// TIA Portal V20 export
DATA_BLOCK "Config"   // DB102
// stored: Access Published, MemoryReserve 100, Namespace Unit1.Em5
   VAR
      em : "LAF_typeEmConfiguration";   // Configuration of EM Parameters
      axis : Array[1.._.U1EM5_NO_OF_AXES] of DB_ANY;
      moduleAccessPoint : Array[1.._.U1EM5_NO_OF_AXES] of HW_SUBMODULE;
   END_VAR
   VAR RETAIN
      cmNgAndManualInputAxisY : "LBC_typeAxis64PosConfiguration";
      cmMagazineAxisZ : "LBC_typeAxis64PosConfiguration";
      cmNgAndManualInputCylinderUpDown : "LBC_typeTwoWayActuatorConfiguration";
      cmNgAndManualInputVacuum1OnOff : "LBC_typeTwoWayActuatorConfiguration";
      cmNgAndManualInputVacuum2OnOff : "LBC_typeTwoWayActuatorConfiguration";
      cmNgAndManualInputVibrator1OnOff : "LBC_typeTwoWayActuatorConfiguration";
      cmNgAndManualInputVibrator2OnOff : "LBC_typeTwoWayActuatorConfiguration";
      cmMagazineLockCylinderUpDown : "LBC_typeTwoWayActuatorConfiguration";
      cmNgAndManaulInputMagazineElectrodeDetectionSensor : "LBC_typeDigitalSignalConfiguration";
      cmNgAndManualInputMagazineDetectionSensor : "LBC_typeDigitalSignalConfiguration";
      cmNgAndManualInputMagazineFullSensor : "LBC_typeDigitalSignalConfiguration";
      cmNgAndManualInputElectrodeDetectionSensor : "LBC_typeDigitalSignalConfiguration";
      cmMagazineSafetyPinIdlePosition : "LBC_typeDigitalSignalConfiguration";
      cmNgAndManualInputAxisY_TorqueCal : "LER_typeServoTorqueCalConfigruation";
      cmMagazineAxisZ_TorqueCal : "LER_typeServoTorqueCalConfigruation";
   END_VAR
BEGIN
   // axis[1] : cmNgAndManualInputAxisY
   // axis[2] : cmMagazineAxisZ
   // moduleAccessPoint[1] : cmNgAndManualInputAxisY
   // moduleAccessPoint[2] : cmMagazineAxisZ
END_DATA_BLOCK
